{attribute 'qualified_only'}
{attribute 'strict'}
TYPE E_SelectedAnimal :
(
	NONE :=0,
	ELEPHANT :=1,
	LION:= 2,
	TIGER := 3
	
);
END_TYPE

(* stored: Version 1.1.0.1, ProductVersion 3.1.4024.16
   DUT E_SelectedAnimal: Id {7469b03a-519c-43b0-be37-479ad484e4b1} *)
